FUNCTION FC1_Bereken_Snelheid : DINT
VAR_INPUT
	gelezenGewicht : DINT := 0;
END_VAR
VAR
	mid : DINT := 0;
	berekendeSnelheid : DINT := 0;
END_VAR


mid := gelezenGewicht / 5;
berekendeSnelheid := mid * 6;

END_FUNCTION

(* stored: Version 1.1.0.1, ProductVersion 3.1.4024.12
   POU FC1_Bereken_Snelheid: Id {96517e6c-c61b-4dd5-868e-97d2735376b2}, SpecialFunc None *)
